TYPE ST_MasterAxisValue :
STRUCT
	Distance			: LREAL;
	Velocity			: LREAL;
	TPhase1			: LREAL;
	TPhase2			: LREAL;
	Acceleration		: LREAL;
	Deceleration		: LREAL;
	Jerk				: LREAL;
	Idx				: INT:=1;
END_STRUCT
END_TYPE

(* stored: Version 1.1.0.1, ProductVersion 3.1.4024.9
   DUT ST_MasterAxisValue: Id {58e5ddb9-3fac-45e9-8c6d-f60bf087a39a} *)
